PROGRAM POU_readSupvData
VAR
	sNetId: T_AmsNetId := SUPVams.sNetId;	// '5.30.23.91.1.1';
	nPort: T_AmsPort := SUPVams.nPort; 		// 851
	FB_ReadAmsValue_Fp: FB_ReadAmsValue;
	FB_ReadAmsValue_R2: FB_ReadAmsValue;
	FB_ReadAmsValue_R3: FB_ReadAmsValue;
	FB_ReadAmsValue_TReactor: FB_ReadAmsValue;
	FB_ReadAmsValue_YA: FB_ReadAmsValue;
	FB_ReadAmsValue_YAC: FB_ReadAmsValue;
	FB_ReadAmsValue_AGI: FB_ReadAmsValue;
	bFpReadError: BOOL;
	nFpReadErrorId: UDINT;
	bR2ReadError: BOOL;
	nR2ReadErrorId: UDINT;
	bR3ReadError: BOOL;
	nR3ReadErrorId: UDINT;
	bTReactorReadError: BOOL;
	nTReactorReadErrorId: UDINT;
	bYAReadError: BOOL;
	nYAReadErrorId: UDINT;
	bYACReadError: BOOL;
	nYACReadErrorId: UDINT;
	bAGIReadError: BOOL;
	nAGIReadErrorId: UDINT;
END_VAR

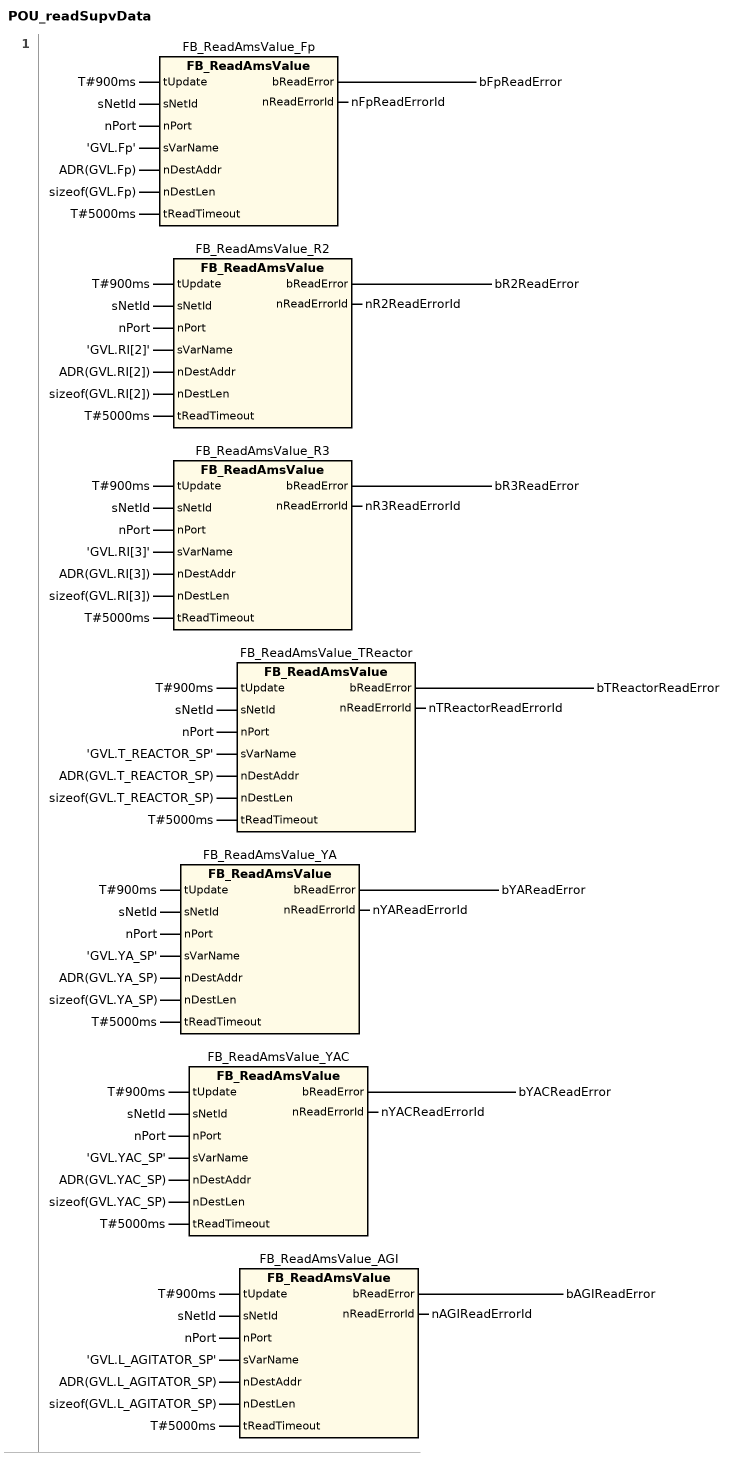
// NETWORK 1
FB_ReadAmsValue_Fp(
    tUpdate := T#900ms,
    sNetId := sNetId,
    nPort := nPort,
    sVarName := 'GVL.Fp',
    nDestAddr := ADR(GVL.Fp),
    nDestLen := sizeof(GVL.Fp),
    tReadTimeout := T#5000ms,
    nReadErrorId => nFpReadErrorId); // FB_ReadAmsValue
bFpReadError := FB_ReadAmsValue_Fp.bReadError;
FB_ReadAmsValue_R2(
    tUpdate := T#900ms,
    sNetId := sNetId,
    nPort := nPort,
    sVarName := 'GVL.RI[2]',
    nDestAddr := ADR(GVL.RI[2]),
    nDestLen := sizeof(GVL.RI[2]),
    tReadTimeout := T#5000ms,
    nReadErrorId => nR2ReadErrorId); // FB_ReadAmsValue
bR2ReadError := FB_ReadAmsValue_R2.bReadError;
FB_ReadAmsValue_R3(
    tUpdate := T#900ms,
    sNetId := sNetId,
    nPort := nPort,
    sVarName := 'GVL.RI[3]',
    nDestAddr := ADR(GVL.RI[3]),
    nDestLen := sizeof(GVL.RI[3]),
    tReadTimeout := T#5000ms,
    nReadErrorId => nR3ReadErrorId); // FB_ReadAmsValue
bR3ReadError := FB_ReadAmsValue_R3.bReadError;
FB_ReadAmsValue_TReactor(
    tUpdate := T#900ms,
    sNetId := sNetId,
    nPort := nPort,
    sVarName := 'GVL.T_REACTOR_SP',
    nDestAddr := ADR(GVL.T_REACTOR_SP),
    nDestLen := sizeof(GVL.T_REACTOR_SP),
    tReadTimeout := T#5000ms,
    nReadErrorId => nTReactorReadErrorId); // FB_ReadAmsValue
bTReactorReadError := FB_ReadAmsValue_TReactor.bReadError;
FB_ReadAmsValue_YA(
    tUpdate := T#900ms,
    sNetId := sNetId,
    nPort := nPort,
    sVarName := 'GVL.YA_SP',
    nDestAddr := ADR(GVL.YA_SP),
    nDestLen := sizeof(GVL.YA_SP),
    tReadTimeout := T#5000ms,
    nReadErrorId => nYAReadErrorId); // FB_ReadAmsValue
bYAReadError := FB_ReadAmsValue_YA.bReadError;
FB_ReadAmsValue_YAC(
    tUpdate := T#900ms,
    sNetId := sNetId,
    nPort := nPort,
    sVarName := 'GVL.YAC_SP',
    nDestAddr := ADR(GVL.YAC_SP),
    nDestLen := sizeof(GVL.YAC_SP),
    tReadTimeout := T#5000ms,
    nReadErrorId => nYACReadErrorId); // FB_ReadAmsValue
bYACReadError := FB_ReadAmsValue_YAC.bReadError;
FB_ReadAmsValue_AGI(
    tUpdate := T#900ms,
    sNetId := sNetId,
    nPort := nPort,
    sVarName := 'GVL.L_AGITATOR_SP',
    nDestAddr := ADR(GVL.L_AGITATOR_SP),
    nDestLen := sizeof(GVL.L_AGITATOR_SP),
    tReadTimeout := T#5000ms,
    nReadErrorId => nAGIReadErrorId); // FB_ReadAmsValue
bAGIReadError := FB_ReadAmsValue_AGI.bReadError;

END_PROGRAM

(* stored: Version 1.1.0.1, ProductVersion 3.1.4024.11
   POU POU_readSupvData: Id {c8dbc9b0-45af-4c0a-8d1c-7f70f78940a5}, SpecialFunc None *)
